RoboDK station: robotics_project_weldingCar.rdk

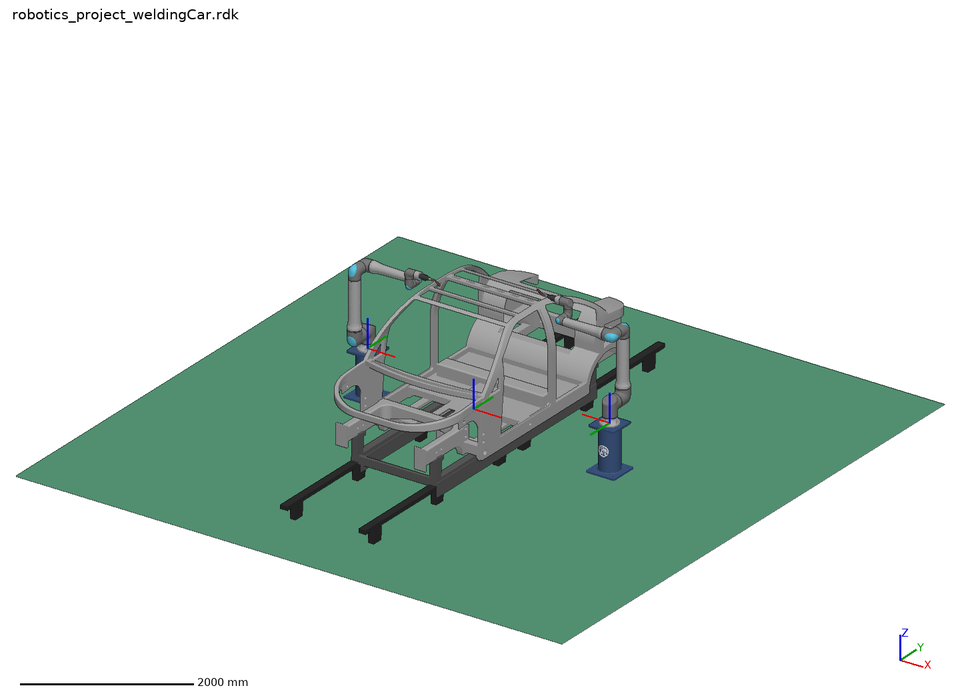
[picture v0: the station drawn from its stored meshes, robots at their saved joint values, targets as dots, program paths as lines]
Station robotics_project_weldingCar (saved by RoboDK 5.9.4). Poses are relative to the parent item; angles as X-Y-Z fixed-axis rotations.
Station parameters (name, value as stored): CollisionFreePlanner, Comau Smart5 NJ 130-2.6, CollisionFreePlanner-Rob Comau Smart5 NJ 130-2.0, CollisionFreePlanner-Rob Comau Smart5 NJ 130-2.6, RoboDK-Comau-RRS1, RoboDK-Comau-RRS1-Backup
  - frame World at (0, 0, 0) mm
    - object Floor at (20, 100, -430) mm, size 7680 x 7680 x 0 mm, geometry from Floor.sld
    - frame Part Reference at (0, 0, 0) mm
      - object Car Frame v24 at (0, 0, 0) mm, size 1740 x 4000 x 1400 mm, geometry from Car Frame v24.step
      - object Car Frame Rack v6 at (0, -1600, -200) mm, size 1260 x 3200 x 510 mm, geometry from Car Frame Rack v6.step
    - object Car Frame Rail v1 at (0, 1480, -230) mm, size 1200 x 6000 x 250 mm
    - frame UR20_LADOA at (-1700, 300, 180) mm
      - robot UR20: 6 axes
          modified DH rows (alpha deg, a mm, theta deg, d mm): 0, 0, 0, 236.2; 90, 0, -180, 0; 0, 861.8, 0, 0; 0, 727.7, 0, 201.9; -90, 0, 0, 159.4; 90, 0, 180, 154.8
          joint limits [-360, -360, -360, -360, -360, -360] to [360, 360, 360, 360, 360, 360]; home [0, -90, -90, 0, 90, 0]; saved at [0, -90, -90, 0, 90, 0]
        - tool Gun, TCP at (89, 0, 340) mm, rotated rx 0 ry 35 rz 0 deg, size 122.1 x 64 x 340.8 mm
    - object Pedestal H24in (Type 1) at (-1700, 300, -430) mm, size 400 x 400 x 609.6 mm, geometry from Pedestal-H24in-Type-1.sld
    - frame UR20_LADOB at (1700, 300, 180) mm, rotated rx 0 ry 0 rz -180 deg
      - robot UR20: 6 axes
          modified DH rows (alpha deg, a mm, theta deg, d mm): 0, 0, 0, 236.2; 90, 0, -180, 0; 0, 861.8, 0, 0; 0, 727.7, 0, 201.9; -90, 0, 0, 159.4; 90, 0, 180, 154.8
          joint limits [-360, -360, -360, -360, -360, -360] to [360, 360, 360, 360, 360, 360]; home [0, -90, -90, 0, 90, 0]; saved at [0, -90, -90, 0, 90, 0]
        - object Gun at (0, 0, 0) mm, size 122.1 x 64 x 340.8 mm
    - object Pedestal H24in (Type 1) at (1700, 300, -430) mm, size 400 x 400 x 609.6 mm, geometry from Pedestal-H24in-Type-1.sld
  - notes Description: <!DOCTYPE HTML PUBLIC "-//W3C//DTD HTML 4.0//EN" "http://www.w3.org/TR/REC-html40/strict.dtd">
<html><head><meta name="qrichtext" content="1" /><meta charset="utf-8" /><style type="text/css">
p, li { white-space: pre-wrap; }
hr { height: 1px; border-width: 0; }
li.unchecked::marker { content: "\2610"; }
li.checked::marker { content: "\2612"; }
</style></head><body style=" font-family:'.AppleSystemUIFont'; font-size:13pt; font-weight:400; font-style:normal;">
<p style=" margin-top:0px; margin-bottom:0px; margin-left:0px; margin-right:0px; -qt-block-indent:0; text-indent:0px;"><span style=" font-family:'MS Shell Dlg 2'; font-size:8.25pt;">This example demonstrates a spot welding application on a full car frame using an industrial 6-axis Comau Smart5 NJ 130-2.6 robot equipped with an OBARA spot welding gun. The goal of this station is to show how RoboDK can be used to create a precise collision-free path within a confined space when using a large welding gun.</span></p></body></html>
